FUNCTION_BLOCK TestLinkedList EXTENDS CNM_Collections.LinkedList
VAR_INPUT
END_VAR
VAR_OUTPUT
END_VAR
VAR
END_VAR

PROPERTY getLastElement : CNM_CollectionInterfaces.IDoublyLinkedElement
GET
getLastElement := THIS^.lastElement;
END_GET
END_PROPERTY

END_FUNCTION_BLOCK

(* stored: Version 1.1.0.1, ProductVersion 3.1.4026.8
   POU TestLinkedList: Id {5d929449-0017-4424-8b61-42864ff2339c}, SpecialFunc None
   Property getLastElement: Id {6b2b38ba-b14b-497f-9e15-b841df61eff8}
   Get Get: Id {4248c1af-4c29-4e19-8ba1-1f25c2304852} *)
